# EPICS substitutions: iocBoot/ioc13ida_linux/MeasCompAliases.substitutions
file "$(CARS)/db/analog_out_alias.template"
{
pattern
{      REC,              ALIAS,                EGUL,  DRVL,  LOPR,  EGUF,  DRVH,  HOPR, PREC,       DESC}
{13IDA:E1608_1:Ao1,  13IDA:CD_MonoPiezoPitch,  -10,     0,      0,   10,    10,    10,    4,   "CD monochromator piezo pitch"}
{13IDA:E1608_1:Ao2,  13IDA:CD_MonoPiezoRoll,   -10,     0,      0,   10,    10,    10,    4,   "CD monochromator piezo roll"}
{13IDA:E1608_2:Ao1,  13IDA:E_MonoPiezoPitch,   -10,     0,    -10,   10,    10,    10,    3,   "E monochromator piezo pitch"}
{13IDA:E1608_2:Ao2,  13IDA:E_MonoPiezoRoll,    -10,     0,    -10,   10,    10,    10,    3,   "E monochromator piezo roll"}
}
